TYPE outWord :
STRUCT
	Lower : USINT; //Lower Bytes
	Upper : USINT; //Upper Bytes
END_STRUCT
END_TYPE

(* stored: Version 1.1.0.1, ProductVersion 3.1.4024.12
   DUT outWord: Id {b8e527f1-62bf-4e11-a722-15ed8cc98432} *)
